INTERFACE ITcoMessageProperties

METHOD Persist : ITcoMessageProperties
END_METHOD

END_INTERFACE

(* stored: Version 1.1.0.1
   Itf ITcoMessageProperties: Id {033ac595-645d-056c-310a-5a8e070f1714}
   Method Persist: Id {54b58622-3387-07ec-2305-491e9eae5e49} *)
